(* IEC 61131-3 sources: festo-codesys-mcp/knowledge/library/utilities, 10 files *)

(* ---- FB_AnalogFilter.st ---- *)
(* =============================================================
   FB_AnalogFilter — First-Order Low-Pass / Moving Average Filter

   Category:     Utilities
   Platform:     CODESYS V3.5 (IEC 61131-3)
   Version:      1.0
   Dependencies: None (standard IEC only)

   Smooths noisy analog signals. Supports two modes:
   - LOW_PASS: Exponential moving average (alpha = tCycle / tFilter)
   - MOVING_AVG: Simple moving average over nSamples

   Usage:
     fbFilter : FB_AnalogFilter;
     fbFilter(rIn := rRawAnalog, nMode := 0, rFilterFactor := 0.1);
     rSmooth := fbFilter.rOut;
   ============================================================= *)
FUNCTION_BLOCK FB_AnalogFilter
VAR_INPUT
    rIn             : REAL;            (* Raw input value *)
    nMode           : INT := 0;        (* 0=Low-pass, 1=Moving average *)
    rFilterFactor   : REAL := 0.1;     (* Low-pass alpha (0.0-1.0, lower=smoother) *)
    nSamples        : INT := 10;       (* Moving average window size (max 32) *)
    bReset          : BOOL;            (* Reset filter to current input *)
END_VAR
VAR_OUTPUT
    rOut            : REAL;            (* Filtered output *)
END_VAR
VAR
    bInit           : BOOL := FALSE;
    (* Moving average buffer *)
    aBuffer         : ARRAY[0..31] OF REAL;
    nIndex          : INT := 0;
    rSum            : REAL := 0.0;
    nCount          : INT := 0;
END_VAR

IF bReset OR NOT bInit THEN
    rOut := rIn;
    bInit := TRUE;
    rSum := 0.0;
    nIndex := 0;
    nCount := 0;
    bReset := FALSE;
END_IF

CASE nMode OF
0: (* Low-pass exponential filter *)
    rOut := rOut + rFilterFactor * (rIn - rOut);

1: (* Moving average *)
    IF nSamples < 1 THEN nSamples := 1; END_IF
    IF nSamples > 32 THEN nSamples := 32; END_IF

    rSum := rSum - aBuffer[nIndex] + rIn;
    aBuffer[nIndex] := rIn;
    nIndex := nIndex + 1;
    IF nIndex >= nSamples THEN
        nIndex := 0;
    END_IF
    IF nCount < nSamples THEN
        nCount := nCount + 1;
    END_IF
    IF nCount > 0 THEN
        rOut := rSum / INT_TO_REAL(nCount);
    END_IF
END_CASE

END_FUNCTION_BLOCK

(* ---- FB_Blink.st ---- *)
(* =============================================================
   FB_Blink — LED/Output Blink Pattern Generator

   Category:     Utilities
   Platform:     CODESYS V3.5 (IEC 61131-3)
   Version:      1.0
   Dependencies: None (standard IEC only)

   Generates a blinking output with configurable on/off times.
   Useful for status LEDs, warning indicators, HMI feedback.

   Usage:
     fbBlink : FB_Blink;
     fbBlink(bEnable := TRUE, tOnTime := T#500MS, tOffTime := T#500MS);
     bLedOutput := fbBlink.bOut;
   ============================================================= *)
FUNCTION_BLOCK FB_Blink
VAR_INPUT
    bEnable     : BOOL;                (* Enable blinking *)
    tOnTime     : TIME := T#500MS;     (* ON duration *)
    tOffTime    : TIME := T#500MS;     (* OFF duration *)
END_VAR
VAR_OUTPUT
    bOut        : BOOL;                (* Blinking output *)
END_VAR
VAR
    tonOn       : TON;
    tonOff      : TON;
END_VAR

IF NOT bEnable THEN
    bOut := FALSE;
    tonOn(IN := FALSE, PT := tOnTime);
    tonOff(IN := FALSE, PT := tOffTime);
    RETURN;
END_IF

IF NOT bOut THEN
    tonOff(IN := TRUE, PT := tOffTime);
    IF tonOff.Q THEN
        bOut := TRUE;
        tonOff(IN := FALSE, PT := tOffTime);
    END_IF
ELSE
    tonOn(IN := TRUE, PT := tOnTime);
    IF tonOn.Q THEN
        bOut := FALSE;
        tonOn(IN := FALSE, PT := tOnTime);
    END_IF
END_IF

END_FUNCTION_BLOCK

(* ---- FB_Debounce.st ---- *)
(* =============================================================
   FB_Debounce — Digital Input Debounce Filter

   Category:     Utilities
   Platform:     CODESYS V3.5 (IEC 61131-3)
   Version:      1.0
   Dependencies: None (standard IEC only)

   Filters noisy digital inputs using a TON timer. Output only
   changes after the input has been stable for tDebounce time.

   Usage:
     fbDebounce : FB_Debounce;
     fbDebounce(bIn := bRawInput, tDebounce := T#50MS);
     bFiltered := fbDebounce.bOut;
   ============================================================= *)
FUNCTION_BLOCK FB_Debounce
VAR_INPUT
    bIn         : BOOL;                (* Raw digital input *)
    tDebounce   : TIME := T#50MS;      (* Debounce time *)
END_VAR
VAR_OUTPUT
    bOut        : BOOL;                (* Filtered output *)
    bRising     : BOOL;                (* Rising edge detected *)
    bFalling    : BOOL;                (* Falling edge detected *)
END_VAR
VAR
    tonOn       : TON;
    tonOff      : TON;
    bPrev       : BOOL;
END_VAR

tonOn(IN := bIn, PT := tDebounce);
tonOff(IN := NOT bIn, PT := tDebounce);

IF tonOn.Q THEN
    bOut := TRUE;
ELSIF tonOff.Q THEN
    bOut := FALSE;
END_IF

bRising  := bOut AND NOT bPrev;
bFalling := NOT bOut AND bPrev;
bPrev    := bOut;

END_FUNCTION_BLOCK

(* ---- FB_DelayedOutput.st ---- *)
(* =============================================================
   FB_DelayedOutput — Output with Post-Run Timer

   Category:     Utilities
   Platform:     CODESYS V3.5 (IEC 61131-3)
   Version:      1.0
   Dependencies: None (standard IEC only)

   Generic output controller that stays ON while the trigger
   is active and continues for a configurable delay after the
   trigger turns off. Common use cases: exhaust fans, cooling
   pumps, lubrication systems, or any output requiring a
   post-operation run-on period.

   Includes thermal overload detection and manual override.

   Usage:
     fbFan : FB_DelayedOutput;
     fbFan(
       bEnable    := TRUE,
       bTrigger   := bProcessActive,
       tPostDelay := T#30S
     );
     bOutput := fbFan.bOutput;
   ============================================================= *)
FUNCTION_BLOCK FB_DelayedOutput
VAR_INPUT
    bEnable             : BOOL := TRUE;     (* Enable output system *)
    bTrigger            : BOOL;             (* Trigger signal — output ON while active *)
    bManualOn           : BOOL;             (* Manual override ON *)
    tPostDelay          : TIME := T#30S;    (* Post-trigger delay *)
    bFeedbackOK         : BOOL := TRUE;     (* Feedback OK — e.g. thermal overload relay *)
END_VAR
VAR_OUTPUT
    bOutput             : BOOL;             (* Output command *)
    bActive             : BOOL;             (* Output running *)
    bPostRun            : BOOL;             (* Post-run phase active *)
    bFeedbackFault      : BOOL;             (* Feedback fault alarm *)
END_VAR
VAR
    tonPostRun          : TON;              (* Post-run timer *)
    bWasTrigger         : BOOL;             (* Previous trigger state *)
    bPostRunning        : BOOL;             (* Post-run in progress *)
END_VAR

IF NOT bEnable THEN
    bOutput := FALSE;
    bActive := FALSE;
    bPostRun := FALSE;
    bFeedbackFault := FALSE;
    bPostRunning := FALSE;
    RETURN;
END_IF;

(* ============================================================
   FEEDBACK PROTECTION
   ============================================================ *)

bFeedbackFault := NOT bFeedbackOK;

(* ============================================================
   POST-RUN LOGIC
   ============================================================ *)

(* Detect trigger turn-off edge *)
IF bWasTrigger AND NOT bTrigger THEN
    bPostRunning := TRUE;
END_IF;
bWasTrigger := bTrigger;

(* Post-run timer *)
tonPostRun(IN := bPostRunning, PT := tPostDelay);
IF tonPostRun.Q THEN
    bPostRunning := FALSE;
    tonPostRun(IN := FALSE);
END_IF;

bPostRun := bPostRunning;

(* ============================================================
   OUTPUT
   ============================================================ *)

(* Output ON when:
   - Trigger active, OR
   - Post-run timer running, OR
   - Manual override
   AND no feedback fault *)
bOutput := (bTrigger OR bPostRunning OR bManualOn) AND NOT bFeedbackFault;
bActive := bOutput;

END_FUNCTION_BLOCK

(* ---- FB_Hysteresis.st ---- *)
(* =============================================================
   FB_Hysteresis — On/Off Control with Deadband

   Category:     Utilities
   Platform:     CODESYS V3.5 (IEC 61131-3)
   Version:      1.0
   Dependencies: None (standard IEC only)

   Implements hysteresis switching: output turns ON when input
   exceeds rSetpoint + rHysteresis/2, turns OFF when input drops
   below rSetpoint - rHysteresis/2. Prevents oscillation.

   Usage:
     fbHyst : FB_Hysteresis;
     fbHyst(rIn := rTemperature, rSetpoint := 50.0, rHysteresis := 4.0);
     bHeaterOn := fbHyst.bOut;
   ============================================================= *)
FUNCTION_BLOCK FB_Hysteresis
VAR_INPUT
    rIn         : REAL;            (* Process value *)
    rSetpoint   : REAL := 50.0;    (* Target setpoint *)
    rHysteresis : REAL := 4.0;     (* Total hysteresis band *)
    bInvert     : BOOL := FALSE;   (* Invert output logic *)
END_VAR
VAR_OUTPUT
    bOut        : BOOL;            (* Control output *)
END_VAR
VAR
    rHigh       : REAL;
    rLow        : REAL;
END_VAR

rHigh := rSetpoint + rHysteresis / 2.0;
rLow  := rSetpoint - rHysteresis / 2.0;

IF rIn >= rHigh THEN
    bOut := NOT bInvert;
ELSIF rIn <= rLow THEN
    bOut := bInvert;
END_IF
(* Between rLow and rHigh: output retains previous state *)

END_FUNCTION_BLOCK

(* ---- FB_MqttPublisher.st ---- *)
(* =============================================================
   FB_MqttPublisher — Simplified MQTT Publish with Auto-Reconnect

   Category:     Utilities
   Platform:     CODESYS V3.5 (IEC 61131-3)
   Version:      1.0
   Dependencies: None (standard IEC only, MQTT client concept)

   Simplified MQTT publish wrapper that manages broker connection,
   automatic reconnection on disconnect, and message publishing.
   Uses a state machine with configurable reconnect delay.

   Usage:
     fbMqtt : FB_MqttPublisher;
     fbMqtt(bEnable     := TRUE,
            sBrokerAddr := '192.168.1.50',
            nPort       := 1883,
            sTopic      := 'plc/temperature',
            sPayload    := REAL_TO_STRING(rTemp));
     bOK := fbMqtt.bConnected AND fbMqtt.bPublished;
   ============================================================= *)
FUNCTION_BLOCK FB_MqttPublisher
VAR_INPUT
    bEnable         : BOOL;                (* Enable MQTT connection *)
    sBrokerAddr     : STRING(80);          (* MQTT broker IP or hostname *)
    nPort           : UINT := 1883;        (* MQTT broker port *)
    sClientId       : STRING(80) := 'CODESYS_PLC';  (* MQTT client identifier *)
    sTopic          : STRING(255);         (* Publish topic *)
    sPayload        : STRING(255);         (* Message payload *)
    bPublish        : BOOL;                (* Rising edge: trigger publish *)
    nQos            : INT := 0;            (* QoS level: 0, 1, or 2 *)
    bRetain         : BOOL := FALSE;       (* Retain flag *)
    tReconnectDelay : TIME := T#5S;        (* Delay before reconnect attempt *)
    tPublishTimeout : TIME := T#3S;        (* Publish acknowledgment timeout *)
END_VAR
VAR_OUTPUT
    bConnected      : BOOL;                (* Broker connection active *)
    bPublished      : BOOL;                (* Last publish succeeded *)
    bBusy           : BOOL;                (* Operation in progress *)
    bErr            : BOOL;                (* Error occurred *)
    nErrId          : DINT;                (* Error code: 0=none, 1=connect, 2=publish, 3=timeout, 4=disconnect *)
    nPublishCount   : UDINT;               (* Total successful publishes *)
END_VAR
VAR
    nState          : INT := 0;            (* State machine *)
    rtrigPublish    : R_TRIG;              (* Publish edge detection *)
    tonReconnect    : TON;                 (* Reconnect delay timer *)
    tonPubTimeout   : TON;                 (* Publish timeout timer *)
    tonConnTimeout  : TON;                 (* Connection timeout timer *)
    hClient         : DWORD := 0;          (* MQTT client handle *)
    nResult         : DINT;                (* Operation result *)
    bConnLost       : BOOL := FALSE;       (* Connection lost flag *)
    nReconnectCount : UDINT := 0;          (* Reconnection attempts *)
    bPubPending     : BOOL := FALSE;       (* Publish waiting for connection *)
END_VAR

(* ============================================================
   EDGE DETECTION
   ============================================================ *)

rtrigPublish(CLK := bPublish);

(* Capture publish request even if not yet connected *)
IF rtrigPublish.Q THEN
    bPubPending := TRUE;
    bPublished := FALSE;
END_IF

(* ============================================================
   MAIN STATE MACHINE
   ============================================================ *)

CASE nState OF

0: (* IDLE — waiting for enable *)
    bBusy := FALSE;
    bConnected := FALSE;
    bPublished := FALSE;
    bErr := FALSE;
    nErrId := 0;
    bConnLost := FALSE;
    IF bEnable THEN
        nState := 10;
    END_IF

10: (* CONNECTING — establish MQTT connection *)
    bBusy := TRUE;
    bErr := FALSE;
    nErrId := 0;
    (* Placeholder: hClient := MqttConnect(sBrokerAddr, nPort, sClientId, ADR(nResult)); *)
    tonConnTimeout(IN := TRUE, PT := T#10S);
    IF tonConnTimeout.Q THEN
        tonConnTimeout(IN := FALSE, PT := T#10S);
        bErr := TRUE;
        nErrId := 1;  (* Connection failed *)
        nState := 70;  (* Go to reconnect wait *)
        RETURN;
    END_IF

    (* Simulated: assume connection established *)
    IF TRUE THEN
        hClient := 1;
        bConnected := TRUE;
        bBusy := FALSE;
        tonConnTimeout(IN := FALSE, PT := T#10S);
        nState := 20;
    END_IF

20: (* CONNECTED — monitor connection, wait for publish *)
    IF NOT bEnable THEN
        nState := 80;
        RETURN;
    END_IF

    (* Check connection health *)
    (* Placeholder: bConnLost := NOT MqttIsConnected(hClient); *)
    IF bConnLost THEN
        bConnected := FALSE;
        nErrId := 4;  (* Disconnect detected *)
        nState := 70;  (* Go to reconnect *)
        RETURN;
    END_IF

    (* Process pending publish *)
    IF bPubPending THEN
        nState := 30;
    END_IF

30: (* PUBLISHING — send MQTT message *)
    bBusy := TRUE;
    (* Placeholder: nResult := MqttPublish(hClient, sTopic, sPayload, nQos, bRetain); *)
    tonPubTimeout(IN := TRUE, PT := tPublishTimeout);

    IF tonPubTimeout.Q THEN
        tonPubTimeout(IN := FALSE, PT := tPublishTimeout);
        bErr := TRUE;
        nErrId := 3;  (* Publish timeout *)
        bPubPending := FALSE;
        bBusy := FALSE;
        nState := 20;
        RETURN;
    END_IF

    (* Simulated: assume publish succeeded *)
    IF TRUE THEN
        bPublished := TRUE;
        bPubPending := FALSE;
        nPublishCount := nPublishCount + 1;
        tonPubTimeout(IN := FALSE, PT := tPublishTimeout);
        bBusy := FALSE;
        bErr := FALSE;
        nErrId := 0;
        nState := 20;
    END_IF

70: (* RECONNECT WAIT — delay before retry *)
    bConnected := FALSE;
    bBusy := TRUE;

    IF NOT bEnable THEN
        nState := 80;
        RETURN;
    END_IF

    tonReconnect(IN := TRUE, PT := tReconnectDelay);
    IF tonReconnect.Q THEN
        tonReconnect(IN := FALSE, PT := tReconnectDelay);
        nReconnectCount := nReconnectCount + 1;
        bConnLost := FALSE;
        nState := 10;  (* Retry connection *)
    END_IF

80: (* DISCONNECT — clean shutdown *)
    IF hClient <> 0 THEN
        (* Placeholder: MqttDisconnect(hClient); *)
        hClient := 0;
    END_IF
    bConnected := FALSE;
    bBusy := FALSE;
    bPubPending := FALSE;
    nState := 0;

END_CASE

END_FUNCTION_BLOCK

(* ---- FB_PidController.st ---- *)
(* =============================================================
   FB_PidController — Generic PID Controller with Anti-Windup

   Category:     Utilities
   Platform:     CODESYS V3.5 (IEC 61131-3)
   Version:      1.0
   Dependencies: None (standard IEC only)

   General-purpose PID controller for any closed-loop control:
   temperature, pressure, flow, position, speed, etc.
   Features: P-I-D action, configurable deadband, output
   clamping, integral anti-windup, and self-retriggering
   cycle timer for consistent sample rate.

   Usage:
     fbPid : FB_PidController;
     fbPid(
       bEnable   := bControlActive,
       rSetpoint := 100.0,
       rFeedback := rSensorValue,
       rKp       := 2.0,
       rKi       := 0.5,
       rKd       := 0.1
     );
     rControlOutput := fbPid.rOutput;
   ============================================================= *)
FUNCTION_BLOCK FB_PidController
VAR_INPUT
    bEnable             : BOOL;             (* Enable control loop *)
    rSetpoint           : REAL;             (* Target value [engineering units] *)
    rFeedback           : REAL;             (* Actual value [engineering units] *)
    (* Tuning parameters *)
    rKp                 : REAL := 1.0;      (* Proportional gain *)
    rKi                 : REAL := 0.0;      (* Integral gain *)
    rKd                 : REAL := 0.0;      (* Derivative gain *)
    (* Output limits *)
    rOutputMax          : REAL := 100.0;    (* Max output *)
    rOutputMin          : REAL := 0.0;      (* Min output *)
    rDeadband           : REAL := 0.0;      (* Error deadband [engineering units] *)
    (* Sample time *)
    tCycleTime          : TIME := T#10MS;   (* Match to PLC task cycle *)
END_VAR
VAR_OUTPUT
    rOutput             : REAL;             (* Control output *)
    bAtSetpoint         : BOOL;             (* Within deadband *)
    rError              : REAL;             (* Current error *)
    bSaturated          : BOOL;             (* Output at limits *)
END_VAR
VAR
    (* PID internal state *)
    rIntegral           : REAL;
    rPrevError          : REAL;
    rDerivative         : REAL;
    (* Calculated terms *)
    rPropTerm           : REAL;
    rIntTerm            : REAL;
    rDerTerm            : REAL;
    rRawOutput          : REAL;
    (* Timing *)
    tonCycle            : TON;
    rDtSeconds          : REAL;
    (* Anti-windup *)
    rIntegralMax        : REAL;
    rIntegralMin        : REAL;
    (* First scan flag *)
    bFirstCycle         : BOOL := TRUE;
END_VAR

(* ============================================================
   CYCLE TIMING — self-retriggering for consistent sample rate
   ============================================================ *)

tonCycle(IN := NOT tonCycle.Q, PT := tCycleTime);
rDtSeconds := TIME_TO_REAL(tCycleTime) / 1000.0;

(* ============================================================
   PID CALCULATION
   ============================================================ *)

IF bEnable THEN
    IF tonCycle.Q OR bFirstCycle THEN
        bFirstCycle := FALSE;

        (* --- Error Calculation --- *)
        rError := rSetpoint - rFeedback;

        (* Deadband: suppress control action near setpoint *)
        IF rDeadband > 0.0 AND ABS(rError) <= rDeadband THEN
            rError := 0.0;
            bAtSetpoint := TRUE;
        ELSE
            bAtSetpoint := FALSE;
        END_IF;

        (* --- Proportional Term --- *)
        rPropTerm := rKp * rError;

        (* --- Integral Term with Anti-Windup --- *)
        IF NOT bSaturated THEN
            rIntegral := rIntegral + (rError * rDtSeconds);
        END_IF;

        (* Clamp integral *)
        IF rKi > 0.0 THEN
            rIntegralMax := (rOutputMax - rOutputMin) / rKi;
        ELSE
            rIntegralMax := 1000.0;
        END_IF;
        rIntegralMin := -rIntegralMax;

        IF rIntegral > rIntegralMax THEN
            rIntegral := rIntegralMax;
        ELSIF rIntegral < rIntegralMin THEN
            rIntegral := rIntegralMin;
        END_IF;

        rIntTerm := rKi * rIntegral;

        (* --- Derivative Term --- *)
        IF rDtSeconds > 0.0 THEN
            rDerivative := (rError - rPrevError) / rDtSeconds;
        ELSE
            rDerivative := 0.0;
        END_IF;
        rDerTerm := rKd * rDerivative;

        rPrevError := rError;

        (* --- Total Output --- *)
        rRawOutput := rPropTerm + rIntTerm + rDerTerm;

        (* --- Output Clamping --- *)
        IF rRawOutput > rOutputMax THEN
            rOutput := rOutputMax;
            bSaturated := TRUE;
        ELSIF rRawOutput < rOutputMin THEN
            rOutput := rOutputMin;
            bSaturated := TRUE;
        ELSE
            rOutput := rRawOutput;
            bSaturated := FALSE;
        END_IF;
    END_IF;
ELSE
    (* --- Disabled: reset all state --- *)
    rOutput := 0.0;
    rIntegral := 0.0;
    rPrevError := 0.0;
    rDerivative := 0.0;
    bFirstCycle := TRUE;
    bAtSetpoint := FALSE;
    bSaturated := FALSE;
END_IF;

END_FUNCTION_BLOCK

(* ---- FB_ScaleInt.st ---- *)
(* =============================================================
   FB_ScaleInt — Linear INT Value Scaling

   Category:     Utilities
   Platform:     CODESYS V3.5 (IEC 61131-3)
   Version:      1.0
   Dependencies: None (standard IEC only)

   Maps an input INT from one range to another. Internal
   calculation uses REAL to avoid integer overflow.

   Usage:
     fbScale : FB_ScaleInt;
     fbScale(nIn := nAdcRaw, nInMin := 0, nInMax := 4095,
             nOutMin := 0, nOutMax := 1000);
     nEngValue := fbScale.nOut;
   ============================================================= *)
FUNCTION_BLOCK FB_ScaleInt
VAR_INPUT
    nIn     : INT;             (* Input value *)
    nInMin  : INT := 0;       (* Input range minimum *)
    nInMax  : INT := 4095;    (* Input range maximum *)
    nOutMin : INT := 0;       (* Output range minimum *)
    nOutMax : INT := 1000;    (* Output range maximum *)
    bClamp  : BOOL := TRUE;   (* Clamp output to OutMin..OutMax *)
END_VAR
VAR_OUTPUT
    nOut    : INT;             (* Scaled output *)
    bErr  : BOOL;            (* Division by zero *)
END_VAR
VAR
    rTemp   : REAL;
    nRange  : INT;
END_VAR

nRange := nInMax - nInMin;
IF nRange = 0 THEN
    bErr := TRUE;
    nOut := nOutMin;
    RETURN;
END_IF

bErr := FALSE;
rTemp := INT_TO_REAL(nIn - nInMin) / INT_TO_REAL(nRange)
         * INT_TO_REAL(nOutMax - nOutMin) + INT_TO_REAL(nOutMin);
nOut := REAL_TO_INT(rTemp);

IF bClamp THEN
    IF nOut > nOutMax THEN nOut := nOutMax;
    ELSIF nOut < nOutMin THEN nOut := nOutMin;
    END_IF
END_IF

END_FUNCTION_BLOCK

(* ---- FB_ScaleReal.st ---- *)
(* =============================================================
   FB_ScaleReal — Linear REAL Value Scaling

   Category:     Utilities
   Platform:     CODESYS V3.5 (IEC 61131-3)
   Version:      1.0
   Dependencies: None (standard IEC only)

   Maps an input REAL from one range to another using linear
   interpolation. Optionally clamps output to limits.

   Usage:
     fbScale : FB_ScaleReal;
     fbScale(rIn := rRawAdc, rInMin := 0.0, rInMax := 32767.0,
             rOutMin := 0.0, rOutMax := 100.0, bClamp := TRUE);
     rPercent := fbScale.rOut;
   ============================================================= *)
FUNCTION_BLOCK FB_ScaleReal
VAR_INPUT
    rIn     : REAL;                (* Input value *)
    rInMin  : REAL := 0.0;        (* Input range minimum *)
    rInMax  : REAL := 32767.0;    (* Input range maximum *)
    rOutMin : REAL := 0.0;        (* Output range minimum *)
    rOutMax : REAL := 100.0;      (* Output range maximum *)
    bClamp  : BOOL := TRUE;       (* Clamp output to OutMin..OutMax *)
END_VAR
VAR_OUTPUT
    rOut    : REAL;                (* Scaled output *)
    bErr  : BOOL;               (* Division by zero (InMax = InMin) *)
END_VAR
VAR
    rRange  : REAL;
END_VAR

rRange := rInMax - rInMin;
IF ABS(rRange) < 1.0E-10 THEN
    bErr := TRUE;
    rOut := rOutMin;
    RETURN;
END_IF

bErr := FALSE;
rOut := (rIn - rInMin) / rRange * (rOutMax - rOutMin) + rOutMin;

IF bClamp THEN
    IF rOut > rOutMax THEN rOut := rOutMax;
    ELSIF rOut < rOutMin THEN rOut := rOutMin;
    END_IF
END_IF

END_FUNCTION_BLOCK

(* ---- FB_Totalizer.st ---- *)
(* =============================================================
   FB_Totalizer — Flow/Energy Integrator with Reset

   Category:     Utilities
   Platform:     CODESYS V3.5 (IEC 61131-3)
   Version:      1.0
   Dependencies: None (standard IEC only)

   Integrates a rate value over time (e.g., liters/min → total liters,
   kW → kWh). Uses trapezoidal integration for accuracy.

   Usage:
     fbTotal : FB_Totalizer;
     fbTotal(bEnable := TRUE, rRate := rFlowLitersPerMin,
             tCycleTime := T#100MS, bReset := FALSE);
     rTotalLiters := fbTotal.rTotal;
   ============================================================= *)
FUNCTION_BLOCK FB_Totalizer
VAR_INPUT
    bEnable     : BOOL;                (* Enable integration *)
    rRate       : REAL := 0.0;         (* Rate value [units/time_base] *)
    tCycleTime  : TIME := T#100MS;     (* PLC scan cycle time *)
    rTimeBase   : REAL := 60.0;        (* Rate time base in seconds (60=per minute) *)
    bReset      : BOOL;                (* Reset total to zero *)
END_VAR
VAR_OUTPUT
    rTotal      : REAL := 0.0;         (* Accumulated total *)
    rPeakRate   : REAL := 0.0;         (* Peak rate recorded *)
END_VAR
VAR
    rPrevRate   : REAL := 0.0;
    rDtSec      : REAL;
END_VAR

IF bReset THEN
    rTotal := 0.0;
    rPeakRate := 0.0;
    rPrevRate := 0.0;
    RETURN;
END_IF

IF NOT bEnable THEN
    rPrevRate := rRate;
    RETURN;
END_IF

(* Convert cycle time to seconds *)
rDtSec := TIME_TO_REAL(tCycleTime) / 1000.0;

(* Trapezoidal integration: average of current and previous rate *)
IF rTimeBase > 0.0 THEN
    rTotal := rTotal + ((rRate + rPrevRate) / 2.0) * (rDtSec / rTimeBase);
END_IF

(* Track peak *)
IF rRate > rPeakRate THEN
    rPeakRate := rRate;
END_IF

rPrevRate := rRate;

END_FUNCTION_BLOCK
